{attribute 'pack_mode' := '2'}
TYPE ST_XPU_CTRL :
STRUCT
  Cmd             : E_XPU_CTRL;
END_STRUCT
END_TYPE

(* stored: Version 1.1.0.1, ProductVersion 3.1.4026.18
   DUT ST_XPU_CTRL: Id {2029cad2-935e-49fd-9fb3-dca5c1ed687a} *)
